FUNCTION_BLOCK TelemetryAccelerometers EXTENDS SM_TelemetryAccelerometers
VAR_INPUT
END_VAR
VAR_OUTPUT
END_VAR
VAR
    _testVar_TelemetryDewpoints : BOOL;
END_VAR

SUPER^(config := config);

END_FUNCTION_BLOCK

(* stored: Version 1.1.0.1, ProductVersion 3.1.4018.5
   POU TelemetryAccelerometers: Id {1f63a301-8918-48e4-9095-5d77aea8bc8c}, SpecialFunc None *)
